{attribute 'qualified_only'}
TYPE E_TrayHollowSelection :
(
	Left,
    Centre,
    Right
)USINT;
END_TYPE

(* stored: Version 1.1.0.1, ProductVersion 3.1.4024.11
   DUT E_TrayHollowSelection: Id {2cb403ce-171c-468d-a92d-984cf0e66bd0} *)
